// Mitsubishi GX Works2 project: 0708-산술곱메모리중복   PLC: Q02/Q02H

PROGRAM MAIN
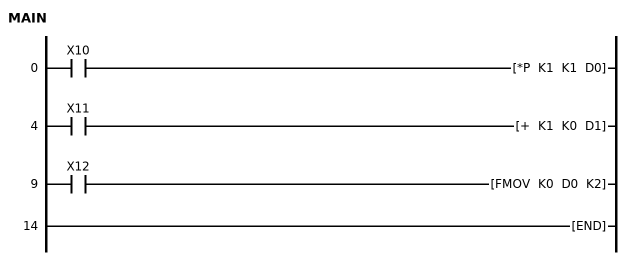
0     LD      X10
      *P      K1 K1 D0
4     LD      X11
      +       K1 K0 D1
9     LD      X12
      FMOV    K0 D0 K2
14    END
END_PROGRAM
